INTERFACE IOnFail EXTENDS __SYSTEM.IQueryInterface

METHOD CarryOn : BOOL
END_METHOD

METHOD Dialog : BOOL
VAR_INPUT
	inRetryStep : INT;
END_VAR
END_METHOD

METHOD DialogWithExternalClose : BOOL
VAR_INPUT
	inRetryStep : INT;
	inRetrySignal:BOOL;
	inTerminateSignal : BOOL;
END_VAR
END_METHOD

METHOD Evaluate : BOOL
VAR_INPUT
	inFromState : INT;
	inFailMode : eTcoInspectorFailMode;
    inToState : INT;
END_VAR
END_METHOD

METHOD Retry : BOOL
VAR_INPUT
	inFromState : INT;
END_VAR
END_METHOD

METHOD RetryThenTerminate : BOOL
VAR_INPUT
	inFromState : INT;
END_VAR
END_METHOD

METHOD Terminate : BOOL
END_METHOD

END_INTERFACE

(* stored: Version 1.1.0.1, ProductVersion 3.1.4024.12
   Itf IOnFail: Id {64413ada-1c4e-0207-0dd6-42d79018c54f}
   Method CarryOn: Id {9390b52f-558b-082c-1e58-cbe248692714}
   Method Dialog: Id {1c9baaa3-a071-0be9-3d2f-47bdb737bd2e}
   Method DialogWithExternalClose: Id {1fb8e24c-a03a-0bc9-33ef-eafe45625661}
   Method Evaluate: Id {3ac67a28-9e55-0b52-3955-5ec6682aa94d}
   Method Retry: Id {35cbf4b9-b3aa-0f5d-0000-a466366ca062}
   Method RetryThenTerminate: Id {f7a58b72-6f87-0c49-0dfe-12fd5d319e9a}
   Method Terminate: Id {6bd31019-9b56-0c3f-1fdb-bb53e3d258fc} *)
